// TIA Portal V19 export
VAR_GLOBAL   // PLC tag table "D04"
   D04_Lp_EntryReq_LB103 AT %Q107.0 : Bool;   // 192SH1
   D04_Lp_SafetyReset_LB103 AT %Q107.1 : Bool;   // 192SH2
   D04_Pb_EntryReq_LB103 AT %I103.4 : Bool;   // 192SH1
   D04_Pb_SafetyReset_LB103 AT %I103.5 : Bool;   // 192SH2
   D04_Unlock AT %Q106.6 : Bool;   // 19202 Comando elettroserratura
   D04_Funzione_AUX_Elettroserratura AT %Q106.7 : Bool;   // 19205
   D04_LockEnable AT %I103.2 : Bool;   // 192A1 cancello chiuso
   D04_Cancello_Bloccato AT %I103.3 : Bool;   // 192A1
   D04_Ls AT %I1020.3 : Bool;   // 102DI3 - 192A1
END_VAR
